PROGRAM MAIN_1
VAR
	pmlbase : PML_Base;
END_VAR

END_PROGRAM

(* stored: Version 1.1.0.1, ProductVersion 3.1.4024.11
   POU MAIN_1: Id {8f22fbc4-6e57-419e-a6c2-cbf5c8ee4798}, SpecialFunc None *)
